// TIA Portal project "FactoryIO_Template_S7-1200_V16_V16" (V16)
// Vorlageprojekt für das Buch mit Zielsystem S7-1200

(* hardware
DEVICE "S7-1200-Station_1"  S7-1200 Station
   slot 0: "Baugruppenträger_0"  Rack  V1.0
   slot 1: "PLC_1"  CPU 1211C DC/DC/DC  6ES7 211-1AE40-0XB0  V4.1
*)

// ===== PLC "PLC_1"  CPU 1211C DC/DC/DC =====

VAR_GLOBAL   // PLC tag table "Standard-Variablentabelle"
   "START FILING" AT %I0.0 : Bool;
   "START DISCHARGE" AT %I0.1 : Bool;
   "FILL VALVE" AT %Q0.0 : Bool;
   "LAMP FILLING" AT %Q0.1 : Bool;
   "DISCHARGE VALVE" AT %Q0.2 : Bool;
   "LAMP DISCHARGE" AT %Q0.3 : Bool;
   "MARKER" AT %M0.0 : Bool;
   "TIMER" AT %QD30 : DInt;
   "MARKER2" AT %M0.1 : Bool;
END_VAR

// folder: System blocks/Program resources

DATA_BLOCK "T1"   // DB1
{ S7_Optimized_Access := 'TRUE' }
AUTHOR : Simatic
FAMILY : IEC
NAME : IEC_TMR
VERSION : 1.0
// stored: InstanceOfName IEC_TIMER
"IEC_TIMER"
BEGIN
END_DATA_BLOCK

DATA_BLOCK "T2"   // DB2
{ S7_Optimized_Access := 'TRUE' }
AUTHOR : Simatic
FAMILY : IEC
NAME : IEC_TMR
VERSION : 1.0
// stored: InstanceOfName IEC_TIMER
"IEC_TIMER"
BEGIN
END_DATA_BLOCK

// folder: (top level)

FUNCTION "MHJ-PLC-Lab-Function-S71200" : Void   // FC9000, SCL
{ S7_Optimized_Access := 'TRUE' }
VERSION : 0.1
   VAR_TEMP
      rdTimeReturn : Int;
      outputTime : DTL;
      SyncVal : Byte;
      forVal : Int;
      forVal_2 : Int;
      Value : Byte;
   END_VAR
   VAR CONSTANT
      CompVal : Byte := 16#34;
      Value_01 : Byte := 16#11;
      Value_01_DW : DWord := 16#A165_D992;
      Value_02_DW : DWord := 16#58BE_4401;
   END_VAR
BEGIN

   #Value:=PEEK(area := 16#82,
        dbNumber := 0,
        byteOffset := 511);
   #Value := #Value + 1;

   POKE(area := 16#82,
        dbNumber := 0,
        byteOffset := 511,
        value := #Value);

   POKE(area:=16#81,
        dbNumber:=0,
        byteOffset:=1016,
        value:=#Value_01_DW);
   POKE(area := 16#81,
        dbNumber := 0,
        byteOffset := 1020,
        value := #Value_02_DW);

   POKE(area := 16#81,
        dbNumber := 0,
        byteOffset := 511,
        value := B#16#00);

   FOR #forVal := 0 TO 120 DO
       FOR #forVal_2:=0 TO 10 DO
           #rdTimeReturn:=RD_SYS_T(#outputTime);
           #rdTimeReturn := WR_SYS_T(#outputTime);
           #rdTimeReturn := RD_SYS_T(#outputTime);
           #rdTimeReturn := WR_SYS_T(#outputTime);
       END_FOR;
       #SyncVal:= PEEK(area := 16#81,
                      dbNumber := 0,
                      byteOffset := 511);
       IF #SyncVal = #CompVal THEN
          GOTO M_1;
       END_IF;
   END_FOR;
   RETURN;

   M_1:
   POKE(area := 16#81,
        dbNumber := 0,
        byteOffset := 511,
        value := B#16#0);
END_FUNCTION

ORGANIZATION_BLOCK "Main"   // OB1, LAD, ProgramCycle
TITLE = "Main Program Sweep (Cycle)"
{ S7_Optimized_Access := 'TRUE' }
VERSION : 0.1
   VAR_INPUT
      Initial_Call : Bool;   // Initial call of this OB
      Remanence : Bool;   // =True, if remanent data are available
   END_VAR
BEGIN

REGION Network 1: Konnektierungsbaustein für PLC-Lab
   // Im Netzwerk 1 wird der Konnektierungsbaustein für PLC-Lab aufgerufen.
   // Dieser Aufruf darf nicht entfernt werden!
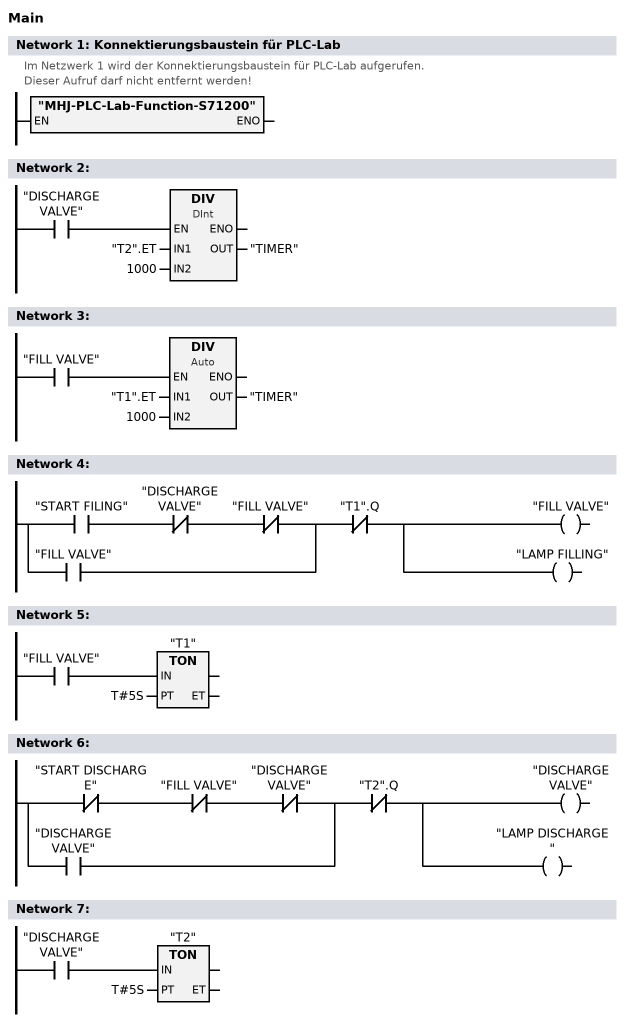
   RUNG wire#powerrail
      "MHJ-PLC-Lab-Function-S71200"()
   END_RUNG
   // the same network as SCL:
   "MHJ-PLC-Lab-Function-S71200"();
END_REGION

REGION Network 2
   RUNG wire#powerrail
      Contact( "DISCHARGE VALVE" )
      { S7_Templates := "SrcType := DInt" } Div(in1 := "T2".ET, in2 := 1000, out => "TIMER")
   END_RUNG
   // the same network as SCL:
   IF "DISCHARGE VALVE" THEN "TIMER" := "T2".ET / 1000; END_IF;
END_REGION

REGION Network 3
   RUNG wire#powerrail
      Contact( "FILL VALVE" )
      Div(in1 := "T1".ET, in2 := 1000, out => "TIMER")
   END_RUNG
   // the same network as SCL:
   IF "FILL VALVE" THEN "TIMER" := "T1".ET / 1000; END_IF;
END_REGION

REGION Network 4
   RUNG wire#powerrail
      Contact( "START FILING" )
      I_Contact( "DISCHARGE VALVE" )
      I_Contact( "FILL VALVE" )
      wire#w1
      I_Contact( "T1".Q )
      wire#w2
      Coil( "FILL VALVE" )
   END_RUNG
   RUNG wire#powerrail
      Contact( "FILL VALVE" )
   END_RUNG wire#w1
   RUNG wire#w2
      Coil( "LAMP FILLING" )
   END_RUNG
   // the same network as SCL:
   "FILL VALVE" := (("START FILING" AND NOT "DISCHARGE VALVE" AND NOT "FILL VALVE") OR "FILL VALVE") AND NOT "T1".Q;
   "LAMP FILLING" := "FILL VALVE";
END_REGION

REGION Network 5
   "T1".TON(IN := "FILL VALVE", PT := T#5S);
END_REGION

REGION Network 6
   RUNG wire#powerrail
      I_Contact( "START DISCHARGE" )
      I_Contact( "FILL VALVE" )
      I_Contact( "DISCHARGE VALVE" )
      wire#w1
      I_Contact( "T2".Q )
      wire#w2
      Coil( "DISCHARGE VALVE" )
   END_RUNG
   RUNG wire#powerrail
      Contact( "DISCHARGE VALVE" )
   END_RUNG wire#w1
   RUNG wire#w2
      Coil( "LAMP DISCHARGE" )
   END_RUNG
   // the same network as SCL:
   "DISCHARGE VALVE" := ((NOT "START DISCHARGE" AND NOT "FILL VALVE" AND NOT "DISCHARGE VALVE") OR "DISCHARGE VALVE") AND NOT "T2".Q;
   "LAMP DISCHARGE" := "DISCHARGE VALVE";
END_REGION

REGION Network 7
   "T2".TON(IN := "DISCHARGE VALVE", PT := T#5S);
END_REGION
END_ORGANIZATION_BLOCK